// Mitsubishi GX Works2 project: PID_program_testing_LL   PLC: FX2N/FX2NC

// task Task_01 (event FALSE, interval T#0.1s, priority 31): LL_ST
// user libraries (not included): basic_lib

FUNCTION_BLOCK SamplingstimeTracker
VAR_INPUT
  ENABLE : BOOL;  (* Activate block *)
  Intervall : TIME;  (* Time between each caluclation *)
END_VAR
VAR_OUTPUT
  SampleTime : REAL;  (* In seconds *)
END_VAR
VAR
  counter : DINT;  (* Increments every cycle *)
  tonFlag : BOOL;
  tonCurrentTIme : TIME;
  time_DINT : DINT;  (* Temporary variable *)
  counter_FLT : REAL;  (* Temporary variable *)
  time_FLT : REAL;  (* Temporary variable *)
  TON_1 : TON;
END_VAR
VAR_INPUT
  warningLimit : REAL;  (* Used for output "warning" *)
END_VAR
VAR_OUTPUT
  warning : BOOL;  (* High if SampleTime > warningLimit *)
END_VAR
(*
	==== 		SampletimeTracker 		====
	

*)

IF ENABLE THEN
	DINC(1, counter);
	TON_1(IN:=1, PT:=Intervall, Q:=tonFlag , ET:=tonCurrentTIme); 			(* Start timer *)
	
	IF tonFlag THEN 
		(* Calculate SampleTime*)
		 time_DINT := TIME_TO_DINT(tonCurrentTIme); 			(* Milliseconds *)
		DFLT(1, time_DINT, time_FLT); 								
		DFLT(1, counter, counter_FLT);
		SampleTime := time_FLT/(counter_FLT*1000.0);
		
		(* Reset variables *)
		TON_1(IN:=0, PT:=Intervall, Q:=tonFlag , ET:=tonCurrentTIme);  		(* Reset timer *)
		counter := 0; 
	END_IF;
	
	(* 	Warning / Alarm *)
	IF SampleTime > warningLimit THEN
		warning := TRUE;	
	END_IF;
	
END_IF;
END_FUNCTION_BLOCK

PROGRAM LL_ST
VAR
  Lead_Lag_ST_1 : Lead_Lag_ST;
  Settpunkt : REAL;
  Padrag : INT;
  Prosessverdi : INT;
  K_ll : REAL;
  Tt : REAL;
  Tn : REAL;
END_VAR
(* structured ladder/FBD written out as ST: instructions are called as NAME(EN, inputs, outputs); _pN, _eN, _tN stand for wires *)
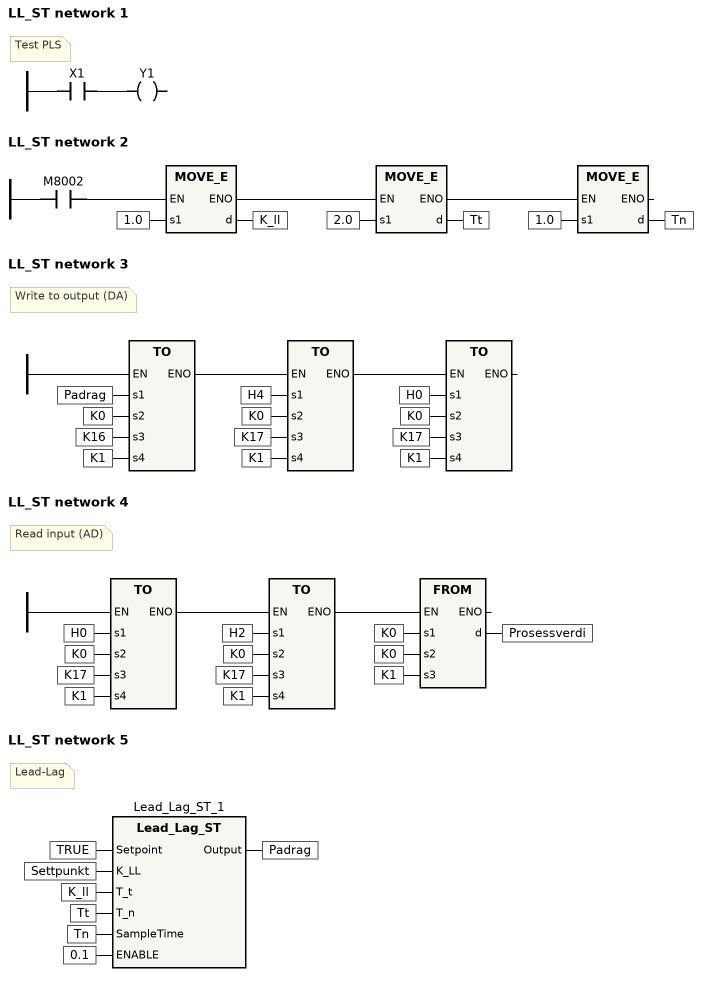
(* network 1 *)
(* Test PLS *)
Y1 := X1;
(* network 2 *)
_e1 := MOVE_E(M8002, 1.0, K_ll);
_e2 := MOVE_E(_e1, 2.0, Tt);
MOVE_E(_e2, 1.0, Tn);
(* network 3 *)
(* Write to output (DA) *)
_e1 := TO(TRUE, Padrag, K0, K16, K1);
_e2 := TO(_e1, H4, K0, K17, K1);
TO(_e2, H0, K0, K17, K1);
(* network 4 *)
(* Read input (AD) *)
_e1 := TO(TRUE, H0, K0, K17, K1);
_e2 := TO(_e1, H2, K0, K17, K1);
FROM(_e2, K0, K0, K1, Prosessverdi);
(* network 5 *)
(* Lead-Lag *)
Lead_Lag_ST_1(Setpoint := TRUE, K_LL := Settpunkt, T_t := K_ll, T_n := Tt, SampleTime := Tn, ENABLE := 0.1, Output => Padrag);
END_PROGRAM

FUNCTION_BLOCK Lead_Lag_ST
VAR_INPUT
  Setpoint : REAL;  (* Settpunkt *)
  K_LL : REAL;  (* Forsterkning til LeadLag *)
  T_t : REAL;  (* Tidskontant teller *)
  T_n : REAL;  (* Tidskonstant nevner *)
  SampleTime : REAL;  (* Tastetid *)
END_VAR
VAR
  LL_Output : REAL;  (* Output pådrag som float *)
END_VAR
VAR_OUTPUT
  Output : INT;  (* Output som enkeltord, for sending til AD/DA *)
END_VAR
VAR_INPUT
  ENABLE : BOOL;
END_VAR
VAR
  U_prev : REAL;  (* Forrige pådag (1 sample tibake) *)
  Setpoint_local : REAL;  (* Lagrer settpunkt til denne variabl *)
  diff1 : REAL;  (* Lagrer utregningene som 3 mellomregninger, for strukutur. *)
  diff2 : REAL;
  diff3 : REAL;
  Setpoint_prev : REAL;  (* Forrige settpunkt(1 sample tilbake) *)
END_VAR
VAR CONSTANT
  MIN_OUTPUT : REAL;  (* Constanter for saturation. *)
  MAX_OUTPUT : REAL := 255.0;
END_VAR

IF ENABLE = 0 THEN
	LL_Output := 0.0;
	Setpoint_local := Setpoint;
ELSE
	Setpoint_local := Setpoint;
	diff1 := Setpoint_prev*K_LL*(SampleTime - 2.0*T_t)/(SampleTime+2.0*T_n);
	diff2 := Setpoint_local*K_LL*(SampleTime+2.0*T_t)/(SampleTime+2.0*T_n);
	diff3 := U_prev*(SampleTime-2.0*T_n)/(SampleTime+2.0*T_n);
	LL_Output := diff1 + diff2 - diff3;
	
	
	(* Saturate both values *)
	IF LL_Output > MAX_OUTPUT THEN                                      
				LL_Output			 := MAX_OUTPUT;
	ELSIF LL_Output < MIN_OUTPUT THEN
				LL_Output 			 := MIN_OUTPUT;
	END_IF;
	
	INT(1, LL_Output,Output);
	
END_IF;
	
U_prev := LL_Output;
Setpoint_prev := Setpoint_local;
END_FUNCTION_BLOCK
